// Brief: Slave Arm MasterSlave controller
FUNCTION_BLOCK PUBLIC FB_SlaveCtrlMasterSlave EXTENDS FB_SlaveArmCtrlBase
VAR_INPUT
END_VAR
VAR_OUTPUT
END_VAR
VAR
END_VAR

METHOD PROTECTED calcCmdJntPos : BOOL
VAR_INPUT
	motionScale :LREAL;
	masterIdx :INT;
END_VAR

VAR_IN_OUT CONSTANT
	i_slaveArm :FB_SlaveArm;
	i_masterStatus :ST_MasterStatus;
END_VAR
VAR 
END_VAR
END_METHOD

// override this function in each exact controller
METHOD PROTECTED calcCmdJntTrq : BOOL
VAR_INPUT
	motionScale :LREAL;
	masterIdx :INT;
END_VAR

VAR_IN_OUT CONSTANT
	i_slaveArm :FB_SlaveArm;
	i_masterStatus :ST_MasterStatus;
END_VAR
VAR 
END_VAR
// set joint torque to zero in default
m_cmdJntTrq := g_zeroVec8d;
END_METHOD

METHOD PUBLIC init : BOOL
VAR_IN_OUT CONSTANT
	i_slaveArm	:FB_SlaveArm;
END_VAR
VAR_IN_OUT 
	r_slaveArmCtrlCmd :ST_SlaveArmCtrlCmds;
END_VAR
SUPER^.Init(i_slaveArm,r_slaveArmCtrlCmd);

m_jntOPMode := g_slaveAllPosTrqMode;
END_METHOD

END_FUNCTION_BLOCK

(* stored: Version 1.1.0.1, ProductVersion 3.1.4024.11
   POU FB_SlaveCtrlMasterSlave: Id {5b96f309-da76-444d-a9fb-2d4321895cd7}, SpecialFunc None
   Method calcCmdJntPos: Id {b549ed00-ec1a-412a-94d0-63a741bf9608}
   Method calcCmdJntTrq: Id {590b7c96-65ed-47d5-8eb2-8a13ee8a5533}
   Method init: Id {1bea1de4-0538-46fc-be44-e671d6da03c3} *)
